(*
Nazwa:			GVL_Checks
Opis:			Zmienne do sprawdzania błędów
Wersja:			v0.1
Data:			2018-10-10
Autor:			DP
Urzadzenia:		
Konfiguracja:	
Info:
(*d*) - obslużone
*)

{attribute 'qualified_only'}
VAR_GLOBAL PERSISTENT
	dCheckBounds		: DINT;	(*Licznik przekroczen zakresu indexow, np. tablic*)
	dCheckDivDInt		: DINT;	(*Licznik prob dzielenia Dint przez 0*)
	dCheckDivLInt		: DINT; (*Licznik prob dzielenia LInt przez 0*)
	dCheckDivLReal		: DINT; (*Licznik prob dzielenia LREAL przez 0*)
	dCheckDivReal		: DINT; (*Licznik prob dzielenia REAL przez 0*)
	dCheckRangeSigned	: DINT;	(*Licznik przekroczen  liczby znakowej*)
	dCheckRangeUnsigned	: DINT; (*Licznik przekroczen  liczby bezznakowej*)
END_VAR

(* stored: Version 1.1.0.1, ProductVersion 3.1.4026.13, FileIdentifier ff6c0b4ef04dab4a61f21da37c4f0adf70560379, FileSignature 1c41a0f42437b5bfb95587e3044347a61200d6dae6b33e9e8dd809dbb657b908d7f9f9baf077d06901dc4e77175643bad9d6c90b8005aa291dc4572646f84dfd8c7f966e1c9b7baa568f8a4663bb0892519726e4954a487d3fc9dc7d73fbff05312663e86dfae9b418eaa4c411bb3261643349987cdf207c2867627023880dc88e177c6109655378babb925414dbd5bfbfbcc9f41e8924d8ba30be99af5e32afa4e5d80a422989bf23e4b482b83dc6d8c47ceffa81a32d440ac0600d34c6f57826a5f84ba33c1baf62f85c3d05771621698e3b6148a5c23fa3a1bd5e2960ccf34b23c3d7142d429ff59c6580f78211038fdf482d31db24f9cb7a91afd7a985a6
   GVL gvlChecks: Id {aa5872d5-628a-4d0d-a807-7ee14c0eb68e} *)
